FUNCTION_BLOCK mergeMsg (* Basic FB with empty ECC *)
  (* Standard: 61499-2 *)
  (* Version 1.0, 2021-03-21, AK120569 *)
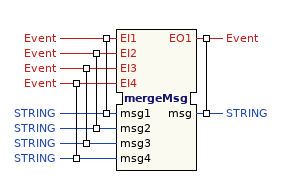
  EVENT_INPUT
    EI1 WITH msg1;
    EI2 WITH msg2;
    EI3 WITH msg3;
    EI4 WITH msg4;
  END_EVENT
  EVENT_OUTPUT
    EO1 WITH msg;
  END_EVENT
  VAR_INPUT
    msg1 : STRING;
    msg2 : STRING;
    msg3 : STRING;
    msg4 : STRING;
  END_VAR
  VAR_OUTPUT
    msg : STRING;
  END_VAR
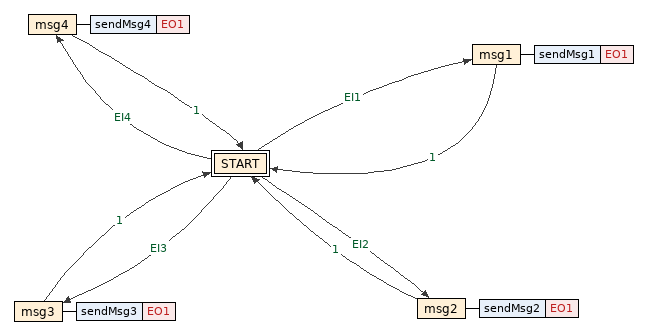
  EC_STATES
    START; (* Initial State *)
    msg2 : sendMsg2 -> EO1;
    msg1 : sendMsg1 -> EO1;
    msg4 : sendMsg4 -> EO1;
    msg3 : sendMsg3 -> EO1;
  END_STATES
  EC_TRANSITIONS
    START TO msg2 := EI2;
    START TO msg1 := EI1;
    START TO msg4 := EI4;
    START TO msg3 := EI3;
    msg3 TO START := 1;
    msg4 TO START := 1;
    msg1 TO START := 1;
    msg2 TO START := 1;
  END_TRANSITIONS
  ALGORITHM sendMsg1 IN ST:
msg := msg1;
  END_ALGORITHM
  ALGORITHM sendMsg2 IN ST:
msg := msg2;
  END_ALGORITHM
  ALGORITHM sendMsg3 IN ST:
msg := msg3;
  END_ALGORITHM
  ALGORITHM sendMsg4 IN ST:
msg := msg4;
  END_ALGORITHM
END_FUNCTION_BLOCK
